FUNCTION WRITE_PROTECTED_ULINT
VAR_INPUT
    Ptr : POINTER TO ULINT;
    Value : ULINT;
END_VAR

Ptr^ := Value;

END_FUNCTION

(* stored: Version 1.1.0.1
   POU WRITE_PROTECTED_ULINT: Id {54c93892-e0bd-4ffb-84a5-c70998b8b8b8}, SpecialFunc None *)
